PROGRAM MAIN
VAR
END_VAR

LightBulbTimer();
Controls();
TankControl();
Alarm_Logic();

END_PROGRAM

(* stored: Version 1.1.0.1, ProductVersion 3.1.4024.9
   POU MAIN: Id {4d780979-07c1-45f9-98b8-995187d5f1f3}, SpecialFunc None *)
